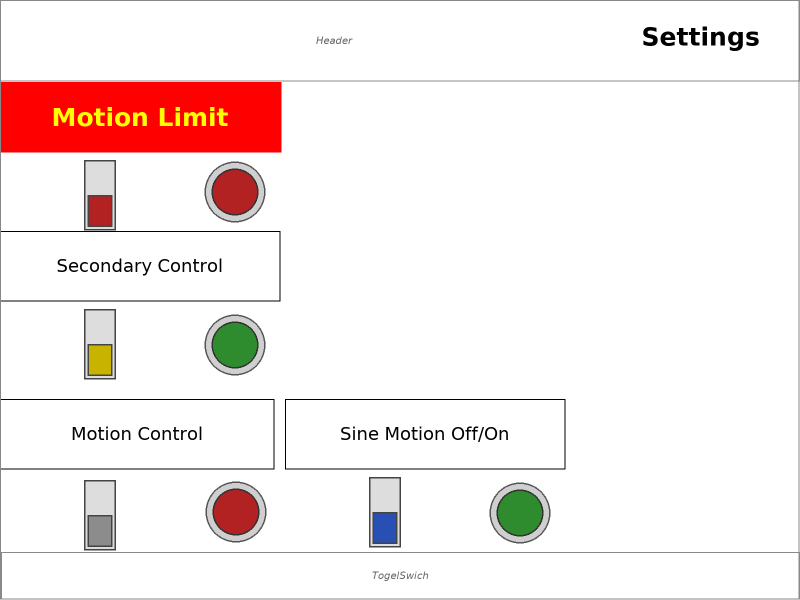
VISUALIZATION Settings  // 800x600
    Rectangle (1,82 280x70), "WARNING"
    Rectangle (0,82 280x70), "Motion Limit", invisible if: HMI.bBlink
    Frame (-132,0 932x81)
        shows Header()
    Frame (1,552 799x47)
        shows TogelSwich()
    Lamp1 (200,157 70x70), variable: HMI.bBlink, style: Lamp-Lamp1-Red
    DipSwitch (20,160 160x70), variable: HMI.bEndStopOverride, behaviour: TOGGLE, style: Switch-DipSwitch-Red
    DipSwitch (20,309 160x70), variable: HMI.bActvateSMC, behaviour: TOGGLE, style: Switch-DipSwitch-Yellow
    Rectangle (0,231 280x70), "Secondary Control"
    Lamp1 (201,477 70x70), variable: HMI.bStartTB, invisible if: not HMI.bStartTB, style: Lamp-Lamp1-Green
    DipSwitch (20,480 160x70), variable: HMI.bStartTB, behaviour: TOGGLE, style: Switch-DipSwitch-Gray
    Rectangle (0,399 274x70), "Motion Control"
    Lamp1 (201,477 70x70), variable: not HMI.bStartTB, invisible if: HMI.bStartTB, style: Lamp-Lamp1-Red
    Lamp1 (200,310 70x70), variable: not HMI.bActvateSMC, style: Lamp-Lamp1-Red
    Textfield (623,20 156x33), "Settings"
    Lamp1 (200,310 70x70), variable: HMI.bActvateSMC, invisible if: not HMI.bActvateSMC, style: Lamp-Lamp1-Green
    DipSwitch (305,477 160x70), variable: HMI.bSwicher, behaviour: TOGGLE, style: Switch-DipSwitch-Blue
    Rectangle (285,399 280x70), "Sine Motion Off/On"
    Lamp1 (485,478 70x70), variable: not HMI.bSwicher, style: Lamp-Lamp1-Red
    Lamp1 (485,478 70x70), variable: HMI.bSwicher, invisible if: not HMI.bSwicher, style: Lamp-Lamp1-Green
END_VISUALIZATION

(* stored: Version 1.1.0.1, ProductVersion 3.1.4024.12
   Visu Settings: Id {c9356fbe-1e1d-4480-8f1a-be136001175e} *)
